Staubli VAL3: progItem.pjx

--- progItem.pjx ---
Parameters version=s7.2.1 stackSize=5000 millimeterUnit=true
Data file=progItem.dtx
Type name=InstrItem path=Disk://kernel/template/InstrItem/InstrItem.pjx

--- progItem.dtx ---
public InstrItem iEvent
  [0]
    string sType
    string sData
public string sID
